(* Common base of all reusable behavior types. *)
FUNCTION_BLOCK ABSTRACT BehaviorBase
VAR_INPUT
	i_params: ParameterSet;
END_VAR
VAR_OUTPUT
	o_status: EOperationResult;
END_VAR
VAR
	(* Because all Control Primitives and Module Sequences instances are 
       singletons, they can set their IDs themselves *)
	m_id: UINT;
	
	(* define's the behavior's parameters (if any)
	   format: <Name1>:<Type1>;<Name2>:<Type2>;... *)
	m_paramDefinition: STRING;
END_VAR

PROPERTY Id : UINT
GET
Id := m_id;
END_GET
END_PROPERTY

PROPERTY ABSTRACT Postcondition : IExpression
GET
END_GET
END_PROPERTY

PROPERTY ABSTRACT Precondition : IExpression
GET
END_GET
END_PROPERTY

END_FUNCTION_BLOCK

(* stored: Version 1.1.0.1, ProductVersion 3.1.4024.9
   POU BehaviorBase: Id {b23e5e53-beeb-455f-9e02-0e5ef5afedb2}, SpecialFunc None
   Property Id: Id {cdaf4337-b8cf-46cc-8218-e52baaed9e34}
   Get Get: Id {cb12a5a4-3bff-4c5b-9b1b-0eb056036a48}
   Property Postcondition: Id {ad8d3d28-609a-449f-897a-feb3e1cc5229}
   Get Get: Id {6dace0f2-c2c6-423f-95ea-cf87e7bfff75}
   Property Precondition: Id {bdc4223a-2a1b-4a81-a2c7-6b9edf536d4a}
   Get Get: Id {e2600cd6-dba1-4c87-b773-83385822a849} *)
